// TIA Portal V20 export
DATA_BLOCK "DB_Analogic_Inputs"   // DB2
{ S7_Optimized_Access := 'TRUE' }
// stored: MemoryReserve 100
   VAR
      Real_Analogic_Input_0 : Real;
      Real_Analogic_Input_1 : Real;
      Uint_Analogic_Input_0 : UInt;
      Uint_Analogic_Input_1 : UInt;
   END_VAR
BEGIN
END_DATA_BLOCK
